Omron CX-Programmer project NewProject (CX-Programmer 9.61)

# PLC NewPLC1: CP1E N30

## Global symbols (name address type ; comment)
0.00 BOOL  ; EMERGENCY STOP
0.01 BOOL  ; START
0.02 BOOL  ; TOMBOL LT 1
0.03 BOOL  ; TOMBOL LT 2
0.04 BOOL  ; TOMBOL LT 3
0.05 BOOL  ; PIL LT 2
0.06 BOOL  ; PILIHAN  LT3
0.07 BOOL  ; PILIHAN LT 1
0.11 BOOL  ; SENSOR LANTAI 1
0.12 BOOL  ; SENSOR LANTAI 2
0.13 BOOL  ; SENSOR LANTAI 3
100.00 BOOL  ; PROSES
100.01 BOOL  ; PINTU LIFT 1
100.02 BOOL  ; PINTU LIFT 2
100.03 BOOL  ; PINTU LIFT 3
101.01 BOOL  ; LAMPU 1
101.02 BOOL  ; LAMPU 2
101.03 BOOL  ; LAMPU 3
103.01 BOOL  ; BUKA LANTAI 1
103.02 BOOL  ; BUKA LANTAI 2
103.03 BOOL  ; BUKA LANTAI 3
105.00 BOOL  ; MOTOR UTAMA
T001 BOOL  ; PINTU 1
T002 BOOL  ; PINTU 2
T003 BOOL  ; PINTU 3
T012 BOOL  ; LANTAI 1 - 2
T013 BOOL  ; LANTAI 1 - 3
T021 BOOL  ; LANTAI 2 - 1
T023 BOOL  ; LANTAI 2 - 3
T031 BOOL  ; LANTAI 3- 1
T032 BOOL  ; LANTAI 3 - 2

## Program NewProgram1 (cyclic task 0)

### Section Section1

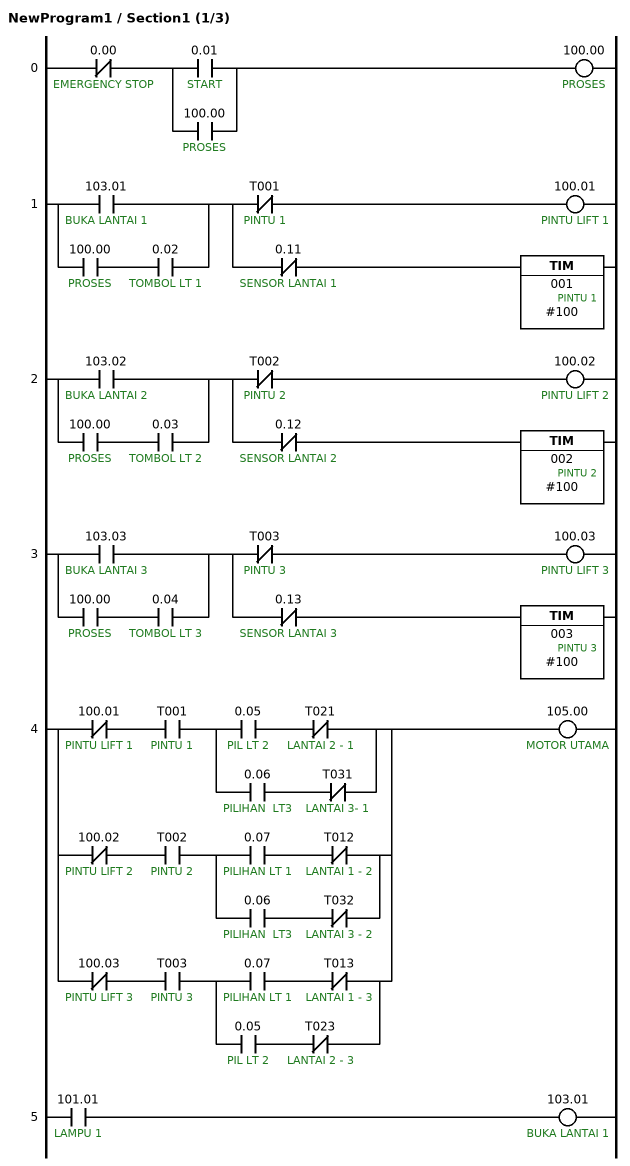
; rung 0
LDNOT 0.00  ; EMERGENCY STOP
LD 0.01  ; START
OR 100.00  ; PROSES
ANDLD
OUT 100.00  ; PROSES
; rung 1
LD 103.01  ; BUKA LANTAI 1
LD 100.00  ; PROSES
AND 0.02  ; TOMBOL LT 1
ORLD
OUT TR0
ANDNOT T001  ; PINTU 1
OUT 100.01  ; PINTU LIFT 1
LD TR0
ANDNOT 0.11  ; SENSOR LANTAI 1
TIM 001 #100  ; PINTU 1
; rung 2
LD 103.02  ; BUKA LANTAI 2
LD 100.00  ; PROSES
AND 0.03  ; TOMBOL LT 2
ORLD
OUT TR0
ANDNOT T002  ; PINTU 2
OUT 100.02  ; PINTU LIFT 2
LD TR0
ANDNOT 0.12  ; SENSOR LANTAI 2
TIM 002 #100  ; PINTU 2
; rung 3
LD 103.03  ; BUKA LANTAI 3
LD 100.00  ; PROSES
AND 0.04  ; TOMBOL LT 3
ORLD
OUT TR0
ANDNOT T003  ; PINTU 3
OUT 100.03  ; PINTU LIFT 3
LD TR0
ANDNOT 0.13  ; SENSOR LANTAI 3
TIM 003 #100  ; PINTU 3
; rung 4
LDNOT 100.01  ; PINTU LIFT 1
AND T001  ; PINTU 1
LD 0.05  ; PIL LT 2
ANDNOT T021  ; LANTAI 2 - 1
LD 0.06  ; PILIHAN  LT3
ANDNOT T031  ; LANTAI 3- 1
ORLD
ANDLD
LDNOT 100.02  ; PINTU LIFT 2
AND T002  ; PINTU 2
LD 0.07  ; PILIHAN LT 1
ANDNOT T012  ; LANTAI 1 - 2
LD 0.06  ; PILIHAN  LT3
ANDNOT T032  ; LANTAI 3 - 2
ORLD
ANDLD
ORLD
LDNOT 100.03  ; PINTU LIFT 3
AND T003  ; PINTU 3
LD 0.07  ; PILIHAN LT 1
ANDNOT T013  ; LANTAI 1 - 3
LD 0.05  ; PIL LT 2
ANDNOT T023  ; LANTAI 2 - 3
ORLD
ANDLD
ORLD
OUT 105.00  ; MOTOR UTAMA
; rung 5
LD 101.01  ; LAMPU 1
OUT 103.01  ; BUKA LANTAI 1

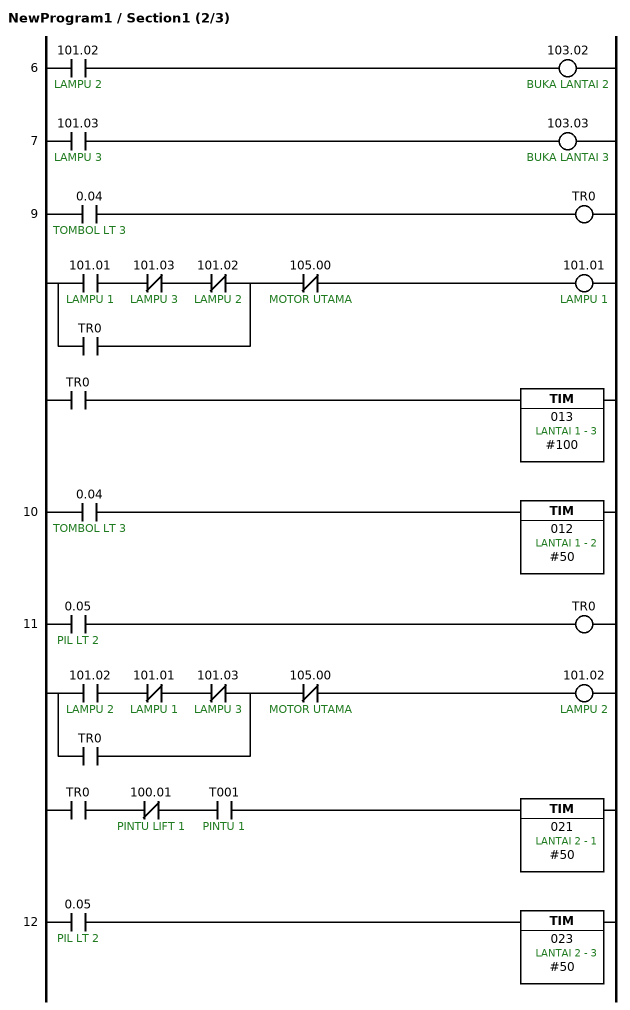
; rung 6
LD 101.02  ; LAMPU 2
OUT 103.02  ; BUKA LANTAI 2
; rung 7
LD 101.03  ; LAMPU 3
OUT 103.03  ; BUKA LANTAI 3
; rung 9
LD 101.01  ; LAMPU 1
ANDNOT 101.03  ; LAMPU 3
ANDNOT 101.02  ; LAMPU 2
LD 0.04  ; TOMBOL LT 3
OUT TR0
ORLD
ANDNOT 105.00  ; MOTOR UTAMA
OUT 101.01  ; LAMPU 1
LD TR0
TIM 013 #100  ; LANTAI 1 - 3
; rung 10
LD 0.04  ; TOMBOL LT 3
TIM 012 #50  ; LANTAI 1 - 2
; rung 11
LD 101.02  ; LAMPU 2
ANDNOT 101.01  ; LAMPU 1
ANDNOT 101.03  ; LAMPU 3
LD 0.05  ; PIL LT 2
OUT TR0
ORLD
ANDNOT 105.00  ; MOTOR UTAMA
OUT 101.02  ; LAMPU 2
LD TR0
ANDNOT 100.01  ; PINTU LIFT 1
AND T001  ; PINTU 1
TIM 021 #50  ; LANTAI 2 - 1
; rung 12
LD 0.05  ; PIL LT 2
TIM 023 #50  ; LANTAI 2 - 3

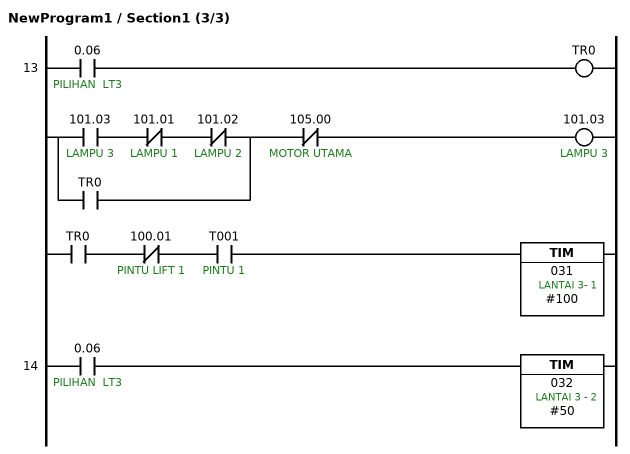
; rung 13
LD 101.03  ; LAMPU 3
ANDNOT 101.01  ; LAMPU 1
ANDNOT 101.02  ; LAMPU 2
LD 0.06  ; PILIHAN  LT3
OUT TR0
ORLD
ANDNOT 105.00  ; MOTOR UTAMA
OUT 101.03  ; LAMPU 3
LD TR0
ANDNOT 100.01  ; PINTU LIFT 1
AND T001  ; PINTU 1
TIM 031 #100  ; LANTAI 3- 1
; rung 14
LD 0.06  ; PILIHAN  LT3
TIM 032 #50  ; LANTAI 3 - 2

### Section END
; rung 0
END(001)